TYPE "Thickness_Par"
VERSION : 0.1
// Block: Thickness_Par
   STRUCT
      SensorON : Bool;
      Trigger_interval : Real;
      NG_Measures_ToFault : Int;
      BypassAutoReset : Int;
      Tolerance_Min : Real;
      Tolerance_Max : Real;
      MES_RecordChange_ThresholdMin : Real;
      MES_RecordChange_ThresholdMax : Real;
   END_STRUCT;

END_TYPE
